// TIA Portal V16 export
// export: Created 2024-12-03T15:41:42.53045Z, ExportSetting WithDefaults, DisplayName Totally Integrated Automation Portal, DisplayVersion V16 Update 6, DisplayName TIA Portal Version Control Interface, DisplayVersion V16 Update 2, DisplayName TIA Portal Openness, DisplayVersion V16 Update 6, DisplayName TIA Portal Teamcenter Gateway, DisplayVersion V16, DisplayName SINAMICS Startdrive Advanced, DisplayVersion V16 Update 5, DisplayName SINAMICS Startdrive G130, G150, S120, S150, SINAMICS MV, S210, DisplayVersion V16 Update 5, DisplayName SINAMICS Startdrive G110M, G120, G120C, G120D, G120P, G115D, DisplayVersion V16 Update 5, DisplayName STEP 7 Professional, DisplayVersion V16 Update 6, DisplayName STEP 7 Safety, DisplayVersion V16, DisplayName WinCC Advanced / Unified PC, DisplayVersion V16 Update 6
FUNCTION_BLOCK "G115D_FB"   // FB48, SCL
{ S7_Optimized_Access := 'TRUE' }
VERSION : 0.1
// stored: AutoNumber true, IsIECCheckEnabled false, IsRetainMemResEnabled false, MemoryReserve 100, SetENOAutomatically false, UDAEnableTagReadback false
   VAR_INPUT
      I_DriveInData : "G115D_INPUT_UDT";
      I_ExtReset : Bool := true;
   END_VAR
   VAR_IN_OUT
      IO_CONTROL : "G115D_OUTPUT_UDT";
      IO_DRIVE : "G115D_DRIVE_UDT";
   END_VAR
   VAR
      cycle : "CycleRun";
      alarm { S7_SetPoint := 'True'} : "AlarmInfo_UDT";
      reset { S7_SetPoint := 'True'} : TOF_TIME;
      turnDriveOff { S7_SetPoint := 'True'} : TOF_TIME;
      disconnected { S7_SetPoint := 'True'} : TON_TIME;
      notOn { S7_SetPoint := 'True'} : TON_TIME;
      AlarmActive : Program_Alarm;
      FaultActive : Program_Alarm;
      FaultDisconnected : Program_Alarm;
      FaultTorqueNok : Program_Alarm;
      FaultTempNok : Program_Alarm;
      FaultCurrentNok : Program_Alarm;
      FaultNotOnTimedOut : Program_Alarm;
      FaultNotReady : Program_Alarm;
      FaultSafetyError : Program_Alarm;
      FaultSto : Program_Alarm;
   END_VAR
   VAR_TEMP
      T_Appstate : "ApplicationState_UDT";
      T_Zone : "ZoneInfo";
      T_On : Bool;
      T_Direction : Bool;
      T_Speed : Real;
      T_Reset : Bool;
   END_VAR
   VAR CONSTANT
      POWER_SUPPLY_OFF : Int := 30016;
   END_VAR
BEGIN
   REGION APPSTATE

       #T_Zone := "ApplicationState_DB".ZoneNames[#IO_DRIVE.Zone];
       #T_Appstate := "ApplicationState_DB".Appstate[#T_Zone.AppStateIndex];

   END_REGION

   REGION DRIVE READY

       #IO_DRIVE.Status.Ready :=
       #I_DriveInData.status.RunningAtSpeed AND
       #I_DriveInData.status.ControlRequest AND
       #I_DriveInData.status.CoastDownActive AND
       #I_DriveInData.status.QuickStopActive;

   END_REGION

   REGION CYCLE COUNTER

       IF "GlobalCycleRunner_FB_DB".O_Cycle = #T_Zone.AppStateIndex THEN
           #cycle();
       END_IF;

   END_REGION

   REGION COMMANDS ALWAYS ON

       #IO_CONTROL.status.ControlByPlc := 1;
       #IO_CONTROL.status.NoCoastDown := 1;
       #IO_CONTROL.status.NoQuickStop := 1;
       #IO_CONTROL.status.EnableRamp := 1;
       #IO_CONTROL.status.EnableContinueRamp := 1;
       #IO_CONTROL.status.EnableSetPoint := 1;

       #IO_CONTROL.status.MotPotSetPointLower := 1;
       #IO_CONTROL.status.MotPotSetPointRaise := 1;

   END_REGION

   REGION COMMANDS

       //Always reset

       #T_On := 0;
       #T_Direction := 0;
       #T_Speed := 0;

       #IO_CONTROL.status.on_off := 0;
       #IO_CONTROL.status.EnableOperation := 0;
       #IO_CONTROL.status.SetPointInversed := 0;
       #IO_CONTROL.setPointSpeed := 0;

       REGION AUTO

           IF #T_Appstate.States.AutoModeActivated.State THEN
               #T_On := #IO_DRIVE.Cmd.OnAuto;
               #T_Direction := #IO_DRIVE.Cmd.DirectionAuto;

               "SetSpeed_FC"(I_SP := #IO_DRIVE.Cmd.SpeedAuto,
          I_Base := #IO_DRIVE.Settings.references.maxSpeedReference,
          I_Max := #IO_DRIVE.Settings.MaxSpeedAuto,
          I_Min := #IO_DRIVE.Settings.MinSpeedAuto,
          O_Res => #T_Speed);

           END_IF;

       END_REGION

       REGION MANUAL

           IF #T_Appstate.States.ManualModeActivated.State THEN

               #T_On := #IO_DRIVE.Cmd.OnManual;

               IF #IO_DRIVE.Settings.AllowManualDirection THEN
                   #T_Direction := #IO_DRIVE.Cmd.DirectionManual;
               ELSE
                   #T_Direction := #IO_DRIVE.Settings.DefaultDirection;
               END_IF;

               "SetSpeed_FC"(I_SP := #IO_DRIVE.Cmd.SpeedManual,
          I_Base := #IO_DRIVE.Settings.references.maxSpeedReference,
          I_Max := #IO_DRIVE.Settings.MaxSpeedManual,
          I_Min := #IO_DRIVE.Settings.MinSpeedManual,
          O_Res => #T_Speed);

           ELSE
               #IO_DRIVE.Cmd.OnManual := 0;
               #IO_DRIVE.Cmd.DirectionManual := 0;
               #IO_DRIVE.Cmd.SpeedManual := 0;
           END_IF;

       END_REGION

       REGION RESET COMMAND ON ERROR 
           // then we don't start after reset :)

           IF #IO_DRIVE.Faults.status > 0 OR NOT #T_Appstate.States.EmergencyOk.State THEN

               #IO_DRIVE.Cmd.OnAuto := 0;
               #IO_DRIVE.Cmd.DirectionAuto := 0;
               #IO_DRIVE.Cmd.SpeedAuto := 0;

               #IO_DRIVE.Cmd.OnManual := 0;
               #IO_DRIVE.Cmd.DirectionManual := 0;
               #IO_DRIVE.Cmd.SpeedManual := 0;

           END_IF;

       END_REGION

       REGION COPY COMMANDS

           IF #IO_DRIVE.Faults.status = 0 AND NOT #IO_DRIVE.Cmd.Interlock AND #T_Appstate.States.EmergencyOk.State THEN
               #IO_CONTROL.status.SetPointInversed := #T_Direction;
               #IO_CONTROL.status.on_off := #T_On;


               "Normalize_Signal_FC"(I_RawData := #T_Speed,
          I_normalizedValue := #IO_DRIVE.Settings.references.referenceSpeed,
          O_Result => #IO_CONTROL.setPointSpeed);

           END_IF;

           #turnDriveOff(IN := #T_On ,
      PT := t#10s,
      Q => #IO_CONTROL.status.EnableOperation);

       END_REGION

   END_REGION

   REGION STATUS

       "DeNormalize_Signal_FC"(I_RawData := #I_DriveInData.Speed,
                               I_normalizedValue := #IO_DRIVE.Settings.references.referenceSpeed,
                               O_Result => #IO_DRIVE.Status.ActualSpeed);

       "DeNormalize_Signal_FC"(I_RawData := #I_DriveInData.Current,
                               I_normalizedValue := #IO_DRIVE.Settings.references.referenceCurrent,
                               O_Result => #IO_DRIVE.Status.Current);

       "DeNormalize_Signal_FC"(I_RawData := #I_DriveInData.Torque,
                               I_normalizedValue := #IO_DRIVE.Settings.references.referenceTorque,
                               O_Result => #IO_DRIVE.Status.Torque);

       #IO_DRIVE.Status.ActualDirection := #T_On AND #T_Direction;

       #IO_DRIVE.Status.CmdRunManualActive := #T_On AND #IO_DRIVE.Status.ManualModeActive;

       #IO_DRIVE.Status.Interlocked := #IO_DRIVE.Cmd.Interlock;

       #IO_DRIVE.Status.ManualCommandsDisabled := NOT #T_Appstate.States.ManualModeActivated.State;
       #IO_DRIVE.Status.ManualModeActive := #T_Appstate.States.ManualModeActivated.State;

       #IO_DRIVE.Status.Running := #I_DriveInData.status.OperationEnabled AND #I_DriveInData.status.Ready;

   END_REGION

   REGION ALARM / FAULT INFO

       IF NOT #alarm.init OR #IO_DRIVE.info.Name = '' THEN
           #IO_DRIVE.info.Name := "buildObjectName"(I_Symbolname := GetSymbolName(variable := #IO_DRIVE, size := 100));
           #alarm.info := "buildAlarmInfo"(I_ObjectName := #IO_DRIVE.info.Name, I_ZoneIndex := #IO_DRIVE.Zone, I_ZoneName := #T_Zone.ZoneName);
           #alarm.init := true;
       END_IF;

   END_REGION

   REGION ALARMS

       #IO_DRIVE.Alarms.AlarmCode := #I_DriveInData.WarnCode;

       REGION ALARM FROM DRIVE X0

           #IO_DRIVE.Alarms.AlarmFromDrive := #I_DriveInData.status.AlarmActive;
           #IO_DRIVE.Alarms.Status.%X0 := #IO_DRIVE.Alarms.AlarmFromDrive;

       END_REGION

       REGION PROGRAM ALARMS

           IF "GlobalCycleRunner_FB_DB".O_Cycle = #T_Zone.AppStateIndex AND #cycle.O_Cycle = 1 THEN

               #AlarmActive(SIG := #IO_DRIVE.Alarms.AlarmFromDrive,
                                SD_1 := #alarm.info,
                                SD_2 := #T_Zone.ZoneName,
                                SD_3 := #IO_DRIVE.info.Name,
                                SD_4 := #IO_DRIVE.Alarms.AlarmCode);

           END_IF;

       END_REGION

       REGION ALARM ACTIVE

           IF #IO_DRIVE.Alarms.Status > 0 THEN
               "ApplicationState_DB".Appstate[#T_Zone.AppStateIndex].Alarms.AlarmActiveInternalPLC := 1;
           END_IF;

       END_REGION

   END_REGION

   REGION FAULTS

       #IO_DRIVE.Faults.FaultCode := #I_DriveInData.FaultCode;

       REGION X0 - FAULT ACTIVE

           IF #I_DriveInData.status.FaultActive  THEN
               #IO_DRIVE.Faults.FaultActive := 1;
           END_IF;

           #IO_DRIVE.Faults.status.%X0 := #IO_DRIVE.Faults.FaultActive;

       END_REGION

       REGION X1 - DISCONNECTED

           #disconnected(IN := NOT #I_DriveInData.status.readyForSwitchOn,
                         PT := t#500ms);

           IF #disconnected.Q OR WORD_TO_INT(#IO_DRIVE.Alarms.AlarmCode) = #POWER_SUPPLY_OFF THEN
               #IO_DRIVE.Faults.Disconnected := 1;
           END_IF;

           #IO_DRIVE.Faults.status.%X1 := #IO_DRIVE.Faults.Disconnected;

       END_REGION

       REGION X2 - TORQUE NOK

           IF NOT #I_DriveInData.status.TorQueOk AND #I_DriveInData.status.readyForSwitchOn THEN
               #IO_DRIVE.Faults.TorqueNOK := 1;
           END_IF;

           #IO_DRIVE.Faults.status.%X2 := #IO_DRIVE.Faults.TorqueNOK;

       END_REGION

       REGION X3 - TEMPERATURE NOK

           IF NOT #I_DriveInData.status.TemperatureOk AND #I_DriveInData.status.readyForSwitchOn THEN
               #IO_DRIVE.Faults.TemperatureNOK := 1;
           END_IF;

           #IO_DRIVE.Faults.status.%X3 := #IO_DRIVE.Faults.TemperatureNOK;

       END_REGION

       REGION X4 - CURRENT NOK

           IF NOT #I_DriveInData.status.CurrentOk AND #I_DriveInData.status.readyForSwitchOn THEN
               #IO_DRIVE.Faults.CurrentNOK := 1;
           END_IF;

           #IO_DRIVE.Faults.status.%X4 := #IO_DRIVE.Faults.CurrentNOK;

       END_REGION

       REGION X5 - NOT ON TIMED OUT

           #notOn(IN := NOT #IO_DRIVE.Status.Running AND #T_On AND NOT #notOn.Q ,
                  PT := t#2000ms);

           IF #notOn.Q  THEN
               #IO_DRIVE.Faults.NotOnTImedOut := 1;
           END_IF;

           #IO_DRIVE.Faults.status.%X5 := #IO_DRIVE.Faults.NotOnTImedOut;

       END_REGION

       REGION X6 - NOT READY

           IF  NOT #IO_DRIVE.Status.Ready AND NOT #IO_DRIVE.Faults.Disconnected THEN
               #IO_DRIVE.Faults.NotReady := 1;
           END_IF;

           #IO_DRIVE.Faults.status.%X6 := #IO_DRIVE.Faults.NotReady;

       END_REGION

       REGION X7 - SAFETY ERROR

           #IO_DRIVE.Faults.status.%X7 := #IO_DRIVE.Faults.SAFETY_ERROR_ACTIVE;

       END_REGION

       REGION X8 - STO ACTIVE

           #IO_DRIVE.Faults.status.%X8 := #IO_DRIVE.Faults.STO_ACTIVE;

       END_REGION

       REGION PROGRAM ALARM

           IF "GlobalCycleRunner_FB_DB".O_Cycle = #T_Zone.AppStateIndex AND #cycle.O_Cycle = 2 THEN

               #FaultActive(SIG := #IO_DRIVE.Faults.FaultActive,
                            SD_1 := #alarm.info,
                            SD_2 := #T_Zone.ZoneName,
                            SD_3 := #IO_DRIVE.info.Name,
                            SD_4 := #IO_DRIVE.Faults.FaultCode);

           END_IF;

           IF "GlobalCycleRunner_FB_DB".O_Cycle = #T_Zone.AppStateIndex AND #cycle.O_Cycle = 3 THEN

               #FaultDisconnected(SIG := #IO_DRIVE.Faults.Disconnected,
                            SD_1 := #alarm.info,
                            SD_2 := #T_Zone.ZoneName,
                            SD_3 := #IO_DRIVE.info.Name);

           END_IF;

           IF "GlobalCycleRunner_FB_DB".O_Cycle = #T_Zone.AppStateIndex AND #cycle.O_Cycle = 4 THEN

               #FaultTorqueNok(SIG := #IO_DRIVE.Faults.TorqueNOK,
                               SD_1 := #alarm.info,
                               SD_2 := #T_Zone.ZoneName,
                               SD_3 := #IO_DRIVE.info.Name);

           END_IF;

           IF "GlobalCycleRunner_FB_DB".O_Cycle = #T_Zone.AppStateIndex AND #cycle.O_Cycle = 5 THEN

               #FaultTempNok(SIG := #IO_DRIVE.Faults.TemperatureNOK,
                             SD_1 := #alarm.info,
                             SD_2 := #T_Zone.ZoneName,
                             SD_3 := #IO_DRIVE.info.Name);

           END_IF;

           IF "GlobalCycleRunner_FB_DB".O_Cycle = #T_Zone.AppStateIndex AND #cycle.O_Cycle = 5 THEN

               #FaultCurrentNok(SIG := #IO_DRIVE.Faults.CurrentNOK,
                                SD_1 := #alarm.info,
                                SD_2 := #T_Zone.ZoneName,
                                SD_3 := #IO_DRIVE.info.Name);

           END_IF;

           IF "GlobalCycleRunner_FB_DB".O_Cycle = #T_Zone.AppStateIndex AND #cycle.O_Cycle = 5 THEN

               #FaultNotOnTimedOut(SIG := #IO_DRIVE.Faults.NotOnTImedOut,
                                   SD_1 := #alarm.info,
                                   SD_2 := #T_Zone.ZoneName,
                                   SD_3 := #IO_DRIVE.info.Name);

           END_IF;

           IF "GlobalCycleRunner_FB_DB".O_Cycle = #T_Zone.AppStateIndex AND #cycle.O_Cycle = 5 THEN

               #FaultNotReady(SIG := #IO_DRIVE.Faults.NotReady,
                              SD_1 := #alarm.info,
                              SD_2 := #T_Zone.ZoneName,
                              SD_3 := #IO_DRIVE.info.Name);

           END_IF;

           IF "GlobalCycleRunner_FB_DB".O_Cycle = #T_Zone.AppStateIndex AND #cycle.O_Cycle = 6 THEN

               #FaultSafetyError(SIG := #IO_DRIVE.Faults.SAFETY_ERROR_ACTIVE,
                              SD_1 := #alarm.info,
                              SD_2 := #T_Zone.ZoneName,
                              SD_3 := #IO_DRIVE.info.Name);

           END_IF;

           IF "GlobalCycleRunner_FB_DB".O_Cycle = #T_Zone.AppStateIndex AND #cycle.O_Cycle = 7 THEN

               #FaultSto(SIG := #IO_DRIVE.Faults.STO_ACTIVE,
                              SD_1 := #alarm.info,
                              SD_2 := #T_Zone.ZoneName,
                              SD_3 := #IO_DRIVE.info.Name);

           END_IF;

       END_REGION

       REGION RESET

           #T_Reset := #IO_DRIVE.Cmd.Reset OR (#T_Appstate.Hmi_Buttons.reset.state.LE AND #I_ExtReset);

           #reset(IN := #T_Reset,
                  PT := t#250ms);

           #IO_CONTROL.status.ackFault := #reset.Q;

           IF #reset.Q THEN
               #IO_DRIVE.Cmd.Reset := 0;

               //Reset faults
               #IO_DRIVE.Faults.FaultActive := 0;
               #IO_DRIVE.Faults.Disconnected := 0;
               #IO_DRIVE.Faults.TorqueNOK := 0;
               #IO_DRIVE.Faults.TemperatureNOK := 0;
               #IO_DRIVE.Faults.CurrentNOK := 0;
               #IO_DRIVE.Faults.NotOnTImedOut := 0;
               #IO_DRIVE.Faults.NotReady := 0;

           END_IF;

       END_REGION

       REGION FAULT ACTIVE

           IF #IO_DRIVE.Faults.status > 0 THEN
               "ApplicationState_DB".Appstate[#T_Zone.AppStateIndex].Alarms.AlarmActiveInternalPLC := 1;
           END_IF;

       END_REGION

   END_REGION
END_FUNCTION_BLOCK
